# EPICS StreamDevice protocol: source/epics/code/simpleRead.proto
Terminator = CR LF;

getVal{
  in "%d";
}
